{attribute 'GeneratedUsingTerminal: EK1122-0000-0018'}
{attribute addProperty BoxType "EK1122-0000-0018"}
{attribute addProperty Id "Beckhoff_EP9xxxsub_EK1100EK1100_AB5A94672A_0001_EP9128_0020_0016A_0001_EP9128_0020_0016_7506857C593"}
{attribute addProperty CRC "3897167155"}
{attribute addProperty Size "595"}
TYPE Beckhoff_EP9xxxEK1122_E84A0D33 EXTENDS EK1122_AB5A9467 :
STRUCT
	{attribute addProperty Name "Beckhoff_EP9xxxsub_EK1100"}
	{attribute addProperty PreviousPort "Beckhoff EP9xxxEK1122 : D"}
	Beckhoff_EP9xxxsub_EK1100 : EK1100_AB5A9467;
	{attribute addProperty Name "A_0001_EP9128_0020_0016"}
	{attribute addProperty PreviousPort "Beckhoff EP9xxxsub EK1100 : C"}
	A_0001_EP9128_0020_0016 : A_0001_EP9128_0020_0016_7506857C;
END_STRUCT
END_TYPE

(* stored: Version 1.2.0.0, ProductVersion 3.1.4024.9
   DUT Beckhoff_EP9xxxEK1122_E84A0D33: Id {474b19b7-1d34-45e9-b9d3-803a4bb3b987} *)
